// TwinCAT 3 PLC project PLC1
// ProgramVersion: 3.1.4022.2
// libraries:
//   ERS_CO2 Payload Decoder, * (PXL-Tech)
//   MSC1608 Payload Decoder, * (PXL-Tech)
//   Tc2_BABasic, * (Beckhoff Automation GmbH)
//   Tc2_EnOcean, * (Beckhoff Automation GmbH)
//   Tc2_Standard, * (Beckhoff Automation GmbH)
//   Tc2_System, * (Beckhoff Automation GmbH)
//   Tc2_TcpIp, * (Beckhoff Automation GmbH)
//   Tc2_Utilities, * (Beckhoff Automation GmbH)
//   Tc3_JsonXml, * (Beckhoff Automation GmbH)
//   Tc3_Module, * (Beckhoff Automation GmbH)
//   VisuSymbols,3.5.10.0,System
// project tree:
//   / GlobalTextList.TcGTLO, PlcTask.TcTTO, Visualization Manager.TcVMO (not stored), VISU_TASK.TcTTO (not stored)
//   GVLs/ GVL1.TcGVL
//   POUs/ EnOcean.TcPOU (not stored), Lichtsturing.TcPOU, MAIN.TcPOU, Beamercontrol.TcPOU
//   VISUs/ Visualization.TcVIS

CONFIGURATION PLC1
    RESOURCE PLC ON TwinCAT3
        TASK PlcTask(INTERVAL := T#10ms, PRIORITY := 6);
        PROGRAM MAIN WITH PlcTask : MAIN;
    END_RESOURCE
END_CONFIGURATION

// ---- GVLs/GVL1.TcGVL
VAR_GLOBAL
	
//lichtsturing
LichtenRAAMKANT AT %Q*: BOOL;
LichtenDEURKANT AT %Q*: BOOL;

AanwezigheidsdetectorRAAMKANT AT %I*: BOOL;
AanwezigheidsdetectorDEURKANT AT %I*: BOOL;

LichtsterkteDEUR AT %I*: INT;
LichtsterkteDEUR2 AT %I*: INT;
LichtsterkteBORD AT %I*: INT;
lichtsterkteBORD2 AT %I*: INT;
LINKERKNOP AT %I* : BOOL;
RECHTERKNOP AT %I* : BOOL;


//beamer & projectorschermsturing

BeamerAANKNOP AT %I* : BOOL;
BeamerUITKNOP AT %I* : BOOL;
Projectorscherm AT %Q* : BOOL;



socketconnectknop AT %I* : BOOL;
socketsendknop AT %I* : BOOL;



//raamsturing


stKL6581            : STR_KL6581;


END_VAR

// ---- POUs/MAIN.TcPOU
PROGRAM MAIN
VAR
END_VAR

Lichtsturing();
EnOcean();
Beamercontrol();

END_PROGRAM

// ---- POUs/Lichtsturing.TcPOU
PROGRAM Lichtsturing
VAR
	timer1: TOF;
	timer2: TOF;
	TP1: TP;
	TP2 : TP;
	TP3 : TP;
	TP4 : TP;
	TP5 :TP;
	TP6 : TP;
	
	bewegingraam : BOOL;
	bewegingdeur : BOOL;
	relaisstandDEUR : BOOL := FALSE;
	relaisstandDEUR_nieuw : BOOL := FALSE;
	relaisstandRAAM : BOOL := FALSE;
	lichtstand2 : BOOL;
	Lichtstand_Prev2: BOOL;
	Lichtstand_Prev: BOOL;
	LichtstatusDEUR : BOOL;
	LichtstatusBORD : BOOL;
	
	

	TONBOOL: BOOL;
	TON1: TON;
	rtrigger: R_TRIG;
	rtrigger2: R_TRIG;
	rtrigger3: R_TRIG;
	rtrigger4: R_TRIG;
	LINKERKNOPULS: BOOL;
	RECHTERKNOPPULS: BOOL;
	relaisstandcheckRAAM: BOOL;
	relaisstandcheckDEUR: BOOL;
	lichtsterktedeurBerekening: INT := 15000;
	lichtsterkteraamBerekening: int := 11000;
	fblicht: FB_Light;
	fblicht2 : FB_light;
	relaisstandraam_nieuw: BOOL;
END_VAR

timer1(IN:=gvl1.AanwezigheidsdetectorRAAMKANT, PT:= T#300S, Q=>bewegingraam, ET=> );
timer2(IN:=gvl1.AanwezigheidsdetectorDEURKANT, PT:= T#300S, Q=>bewegingdeur , ET=> );



fblicht(bOn:= (LichtsterkteDEUR < lichtsterktedeurBerekening AND bewegingdeur = TRUE), 
bOff:= NOT (LichtsterkteDEUR < lichtsterktedeurBerekening AND bewegingdeur = TRUE), 
bToggle:=RECHTERKNOP, bLight=> relaisstandDEUR_nieuw);

IF (relaisstandDEUR = NOT relaisstandDEUR_nieuw) THEN
	TP2.IN := TRUE;
	relaisstandDEUR := relaisstandDEUR_nieuw;
ELSE
	TP2.IN := FALSE;
END_IF


TP2( PT:=T#50MS , Q => GVL1.LichtenDEURKANT);


fblicht2(bOn:= (LichtsterkteBORD < lichtsterkteraamBerekening AND bewegingraam = TRUE), 
bOff:= NOT (LichtsterkteBORD < lichtsterkteraamBerekening AND bewegingraam = TRUE), 
bToggle:=LINKERKNOP, bLight=> relaisstandraam_nieuw);

IF (relaisstandraam = NOT relaisstandraam_nieuw) THEN
	TP1.IN := TRUE;
	relaisstandraam := relaisstandraam_nieuw;
ELSE
	TP1.IN := FALSE;
END_IF


TP1( PT:=T#50MS , Q => GVL1.LichtenRAAMKANT);

END_PROGRAM

// ---- POUs/Beamercontrol.TcPOU
PROGRAM Beamercontrol



VAR
	
	fbsocketsend: FB_SocketSend;
	bconnect AT %I* : BOOL;
	test : int;
	clientserver: FB_ClientServerConnection;


	
	Beamerstand: LINT;
END_VAR


VAR_INPUT

       
nMode           : DWORD := 16#8000000;



 
BeamerON    : LINT := 16#020000000002;
BeamerOFF 	: LINT := 16#020100000003;
beamerINPUTCHANGE : LINT :=16#020300000201060E;


	
	 


      	sSrvNetId       : T_AmsNetId := '5.52.70.129.1.1';
	  
        sRemoteHost     : STRING(15) := '192.168.0.102';
        nRemotePort     : UDINT := 7142;
        bExecute                : BOOL;
        tTimeout                : TIME := T#45S;
		tReconnect      : TIME := T#45S;(*!!!*)
		

//socketsend       
               
        cbLen           : UDINT;                        
        pSrc            : DWORD;    
		            
           
END_VAR  

VAR_OUTPUT
        bBusy           : BOOL;
        bError          : BOOL;
        nErrId          : UDINT;
		nErrId2          : UDINT;
        hSocket        : T_HSOCKET;
		eState          : E_SocketConnectionState := eSOCKET_DISCONNECTED;
		
	
END_VAR

	



clientserver(
	sSrvNetID:= '', 
	nMode:=CONNECT_MODE_ENABLEDBG , 
	sRemoteHost:= sremoteHost , 
	nRemotePort:= nremoteport, 
	bEnable:= bconnect, 
	tReconnect:= tReconnect, 
	bBusy=> bBusy, 
	bError=> berror,
	nErrId=>nErrId , 
	hSocket=>hsocket , 
	eState=> eState);
	
	IF BeamerAANKNOP = TRUE THEN
	
		
		bExecute := TRUE;
		Beamerstand := BeamerON;
	
ELSE
	
	IF BeamerUITKNOP = TRUE THEN
		
		bExecute := TRUE;
		Beamerstand := BeamerOFF;
	ELSE
		
		bExecute := FALSE;
		Beamerstand := 0;
	END_IF
	
	END_IF
	

	
	
	fbsocketsend(
	sSrvNetId:='' , 
	hSocket:= clientserver.hSocket, 
	cbLen:= 50, 
	pSrc:= ADR(Beamerstand), 
	bExecute:= bexecute , 
	tTimeout:=tTimeout , 
	bBusy=> bBusy , 
	bError=> bError, 
	nErrId=> nErrId2);

END_PROGRAM

// ---- GlobalTextList.TcGTLO
TEXTLIST GlobalTextList
  42 = 'Beamer OFF'
  198 = 'Beamer ON'
  787 = 'Deurkant'
  774 = 'Raamkant'
END_TEXTLIST

// ---- VISUs/Visualization.TcVIS
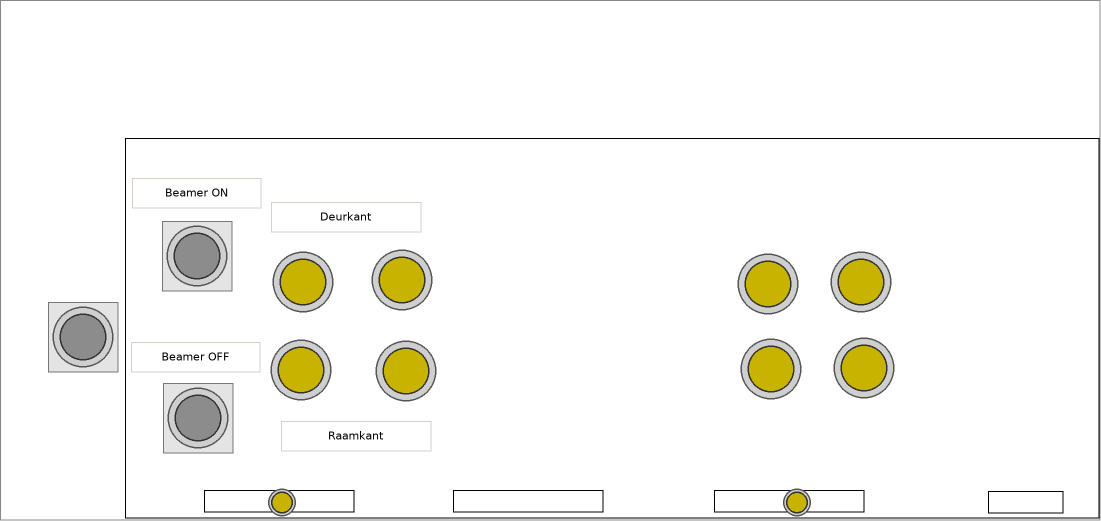
VISUALIZATION Visualization  // 1101x521
    Rectangle (125,138 974x380)
    Lamp1 (268,247 70x70), variable: Lichtsturing.relaisstandDEUR, style: Lamp-Lamp1-Yellow
    Lamp1 (367,245 70x70), variable: Lichtsturing.relaisstandDEUR, style: Lamp-Lamp1-Yellow
    Lamp1 (733,249 70x70), variable: Lichtsturing.relaisstandDEUR, style: Lamp-Lamp1-Yellow
    Lamp1 (826,247 70x70), variable: Lichtsturing.relaisstandDEUR, style: Lamp-Lamp1-Yellow
    Lamp1 (266,335 70x70), variable: Lichtsturing.relaisstandRAAM, style: Lamp-Lamp1-Yellow
    Lamp1 (371,336 70x70), variable: Lichtsturing.relaisstandRAAM, style: Lamp-Lamp1-Yellow
    Lamp1 (736,334 70x70), variable: Lichtsturing.relaisstandRAAM, style: Lamp-Lamp1-Yellow
    Lamp1 (829,333 70x70), variable: Lichtsturing.relaisstandRAAM, style: Lamp-Lamp1-Yellow
    Rectangle (204,490 150x22)
    Rectangle (453,490 150x22)
    Rectangle (714,490 150x22)
    Rectangle (988,491 75x22)
    Lamp1 (266,486 32x33), variable: EnOcean.raam2open, style: Lamp-Lamp1-Yellow
    Lamp1 (781,486 32x33), variable: EnOcean.raam1open, style: Lamp-Lamp1-Yellow
    Textfield (271,202 150x30), "Deurkant"
    Textfield (281,421 150x30), "Raamkant"
    PushSwitch (162,221 70x70), variable: BeamerAANKNOP, behaviour: TOGGLE, style: Switch-PushSwitch-Gray
    Textfield (132,178 129x30), "Beamer ON"
    PushSwitch (163,383 70x70), variable: BeamerUITKNOP, behaviour: TOGGLE, style: Switch-PushSwitch-Gray
    Textfield (131,342 129x30), "Beamer OFF"
    PushSwitch (48,302 70x70), variable: Beamercontrol.bconnect, behaviour: TOGGLE, style: Switch-PushSwitch-Gray
END_VISUALIZATION
